# EPICS substitutions: apps/jscalerApp/Db/wf/jscalers_wf_S4.substitutions
file "db/jscalers_wf_averages-1type-1sector.db" {
pattern { T S }
{ FADC 4 }
{ TRG 4 }
{ TDC 4 }
}
